{attribute 'GeneratedUsingTerminal: AX8206-0100-0101-0101'}
{attribute addProperty BoxType "AX8206-0100-0101-0101"}
{attribute addProperty Id "Ch_B_Target_positionAT %Q*DINT4Ch_B_Target_velocityAT %Q*DINT4"}
{attribute addProperty CRC "4162432626"}
{attribute addProperty Size "8"}
TYPE Ch_B_Interpolator_Outputs_F819AE72 :
STRUCT
	{attribute addProperty Name "Ch_B_Target_position"}
	Ch_B_Target_position AT %Q* : DINT;
	{attribute addProperty Name "Ch_B_Target_velocity"}
	Ch_B_Target_velocity AT %Q* : DINT;
END_STRUCT
END_TYPE

(* stored: Version 1.2.0.0, ProductVersion 3.1.4024.9
   DUT Ch_B_Interpolator_Outputs_F819AE72: Id {e11dab38-8b7f-42d8-af33-f0c76c7a043f} *)
